// Implicitly generated code : DO NOT EDIT
FUNCTION CheckDivLInt : LINT
VAR_INPUT
	divisor:LINT;
END_VAR

// Implicitly generated code : Only an Implementation suggestion
{noflow}
Fault_Count_G(CU:=FALSE) ; 
IF divisor = 0 THEN
	CheckDivLInt:=1;
		Fault_Count_G(CU:=TRUE) ; 
ELSE
	CheckDivLInt:=divisor;
END_IF;
{flow}

END_FUNCTION

(* stored: Version 1.1.0.1, ProductVersion 3.1.4024.2
   POU CheckDivLInt: Id {533d9aeb-a2b8-4b80-bf38-8bb87614be06}, SpecialFunc CheckDivInt64 *)
